// TIA Portal V16 export
// export: Created 2021-09-08T12:46:16.3371185Z, ExportSetting WithDefaults, DisplayName Totally Integrated Automation Portal, DisplayVersion V16 Update 3, DisplayName TIA Portal Version Control Interface, DisplayVersion V16 Update 2, DisplayName TIA Portal Openness, DisplayVersion V16 Update 3, DisplayName TIA Portal Teamcenter Gateway, DisplayVersion V16, DisplayName STEP 7 Professional, DisplayVersion V16 Update 3, DisplayName STEP 7 Safety, DisplayVersion V16, DisplayName WinCC Advanced, DisplayVersion V16 Update 3
TYPE "UF_FLAGS"
// stored: IsFailsafeCompliant false
   STRUCT
      StandBy : Bool;
      Stop : Bool;
      Filtration : Bool;
      Start : Bool;
      HW : Bool;
      HW_A : Bool;
      CEB1 : Bool;
      CEB1_A : Bool;
      CEB2 : Bool;
      CEB2_A : Bool;
      Err : Bool;
      ErrWork : Bool;
      ErrHW : Bool;
      ErrCEB1 : Bool;
      ErrCEB2 : Bool;
      ErrHDP : Bool;
   END_STRUCT;
END_TYPE
